(* IEC 61131-3 sources: pandora_hardware/epos_controller, 7 files *)

(* ---- canRecover.TYP ---- *)
[IEC_IEC_NORM]
TYPE CAN_RECOVER_STATE :(
	CAN_CanError,
	CAN_PowerOffGracefully,
	CAN_Sleep,
	CAN_CanReset,
	CAN_CanReset_loop,
	CAN_SleepWait
) := CAN_CanError;
END_TYPE

(* ---- initial.TYP ---- *)
[IEC_IEC_NORM]
TYPE INITIALIZE_STATE :(
	(*Initialize all axis*)
	INITIALIZE_Init,		(* 0 *)
	(*check the status of axis0*)
	INITIALIZE_CheckAxis0,	(* 1 *)
	(*check the status of axis1*)
	INITIALIZE_CheckAxis1,	(* 2 *)
	(*check the status of axis2*)
	INITIALIZE_CheckAxis2,  (* 3 *)
	(*check the status of axis3*)
	INITIALIZE_CheckAxis3,  (* 4 *)
	(*power of both axis*)
	INITIALIZE_PowerOff,	(* 5 *)
	(*reset axis0*)
	INITIALIZE_Reset0,		(* 6 *)
	(*loop until axis0 is reset*)
	INITIALIZE_Reset0_loop,	(* 7 *)
	(*reset axis1*)
	INITIALIZE_Reset1,		(* 8 *)
	(*wait until axis1 is reset*)
	INITIALIZE_Reset1_loop,	(* 9 *)
	(*reset axis2*)
	INITIALIZE_Reset2,      (* 10 *)
	(*loop until axis2 is reset*)
	INITIALIZE_Reset2_loop, (* 11 *)
	(*reset axis3*)
	INITIALIZE_Reset3,      (* 12 *)
	(*loop until axis3 is reset*)
	INITIALIZE_Reset3_loop, (* 13 *)
	(*power on all axis*)
	INITIALIZE_PowerOn,		(* 14 *)
	(*stop both axis*)
	INITIALIZE_Stop,		(* 15 *)
	(*loop until all axis have stoped*)
	INITIALIZE_Stop_loop,	(* 16 *)
	INITIALIZE_StateHalt0,	(* 17 *)
	INITIALIZE_CanError,    (* 18 *)
	INITIALIZE_CanError_loop(* 19 *)
) := INITIALIZE_Init;
END_TYPE

(* ---- initialize.TYP ---- *)
[IEC_IEC_NORM]
TYPE INITIALIZE_STATE :(
	(*Initialize both axis*)
	INITIALIZE_Init,		(* 0 *)
	(*check the status of axis0*)
	INITIALIZE_CheckAxis0,	(* 1 *)
	(*check the status of axis1*)
	INITIALIZE_CheckAxis1,	(* 2 *)
	(*power of both axis*)
	INITIALIZE_PowerOff,	(* 3 *)
	(*reset axis0*)
	INITIALIZE_Reset0,		(* 4 *)
	(*loop until axis0 is reset*)
	INITIALIZE_Reset0_loop,	(* 5 *)
	(*reset axis1*)
	INITIALIZE_Reset1,		(* 6 *)
	(*wait until axis1 is reset*)
	INITIALIZE_Reset1_loop,	(* 7 *)
	(*power on both axis*)
	INITIALIZE_PowerOn,		(* 8 *)
	(*stop both axis*)
	INITIALIZE_Stop,		(* 9 *)
	(*loop until both axis have stoped*)
	INITIALIZE_Stop_loop,	(* 10 *)
	INITIALIZE_StateHalt0,	(* 11 *)
	INITIALIZE_CanError,
	INITIALIZE_CanError_loop
) := INITIALIZE_Init;
END_TYPE

(* ---- usertype.typ ---- *)
[IEC_IEC_NORM]
TYPE MAIN_STATE :(
	(*initialize all controllers to power on - stand still*)
	(*uses function block FB_INITIALIZE*)
	MAIN_Init,					(* 0 *)
	MAIN_Init_loop,				(* 1 *)

	(*Resets the 3s timeout timer to zero*)
	MAIN_ResetTimer,			(* 2 *)

	(*Reads the control word from EPOS*)
	MAIN_Read,					(* 3 *)
	MAIN_Read_loop,				(* 4 *)

	(*Reads the actual velocity of EPOS P and stores it to a local variable*)
	MAIN_Read_Velocity,			(* 5 *)
	MAIN_Read_Velocity_loop,	(* 6 *)

	(*Reads the actual current of EPOS P and stores it to a local variable*)
	MAIN_Read_Current,			(* 7 *)
	MAIN_Read_Current_loop,		(* 8 *)

	(*Writes the actual velocity of EPOS P from the local variable to EPOS object dictionary*)
	MAIN_Write_Velocity,		(* 9 *)
	MAIN_Write_Velocity_loop,	(* 10 *)

	(*Writes the actual current of EPOS P from the local variable to EPOS object dictionary*)
	MAIN_Write_Current,			(* 11 *)
	MAIN_Write_Current_loop,	(* 12 *)

	(*updatess the timeout timer*)
	(*if the timer reaches 3s switches to state halt*)
	MAIN_UpdateTimer,			(* 13 *)

	(*Executes the move specified by the control word*)
	MAIN_StateAxis_Move,		(* 14 *)

	(*Resets the control word in order to accept a new command*)
	MAIN_StateWrite,			(* 15 *)

	(*halts all motors*)
	MAIN_StateHalt0,			(* 16 *)
	MAIN_StateHalt1,			(* 17 *)

	(*attempts an error recovery if there is CAN error*)
	(*uses function block FB_CanRecover*)
	MAIN_CanError,				(* 18 *)
	MAIN_CanError_loop,			(* 19 *)

	(*Intercepts non-CAN errors coming from other FBs to MAIN_Init*)
	(*uses FB_ErrorWarning to write error codes to EPOS Object Dictionary*)
	MAIN_Error,					(* 20 *)
	MAIN_Error_loop				(* 21 *)
	) := MAIN_Init;
END_TYPE

TYPE INITIALIZE_STATE :(
	(*Initialize both axis*)
	INITIALIZE_Init,		(* 0 *)
	(*check the status of axis0*)
	INITIALIZE_CheckAxis0,	(* 1 *)
	(*check the status of axis1*)
	INITIALIZE_CheckAxis1,	(* 2 *)
	(*check the status of axis2*)
	INITIALIZE_CheckAxis2,  (* 3 *)
	(*check the status of axis3*)
	INITIALIZE_CheckAxis3,  (* 4 *)
	(*power of both axis*)
	INITIALIZE_PowerOff,	(* 5 *)
	(*reset axis0*)
	INITIALIZE_Reset0,		(* 6 *)
	(*loop until axis0 is reset*)
	INITIALIZE_Reset0_loop,	(* 7 *)
	(*reset axis1*)
	INITIALIZE_Reset1,		(* 8 *)
	(*wait until axis1 is reset*)
	INITIALIZE_Reset1_loop,	(* 9 *)
	(*reset axis2*)
	INITIALIZE_Reset2,      (* 10 *)
	(*loop until axis2 is reset*)
	INITIALIZE_Reset2_loop, (* 11 *)
	(*reset axis3*)
	INITIALIZE_Reset3,      (* 12 *)
	(*loop until axis3 is reset*)
	INITIALIZE_Reset3_loop, (* 13 *)
	(*power on all axis*)
	INITIALIZE_PowerOn,		(* 14 *)
	(*stop all axis*)
	INITIALIZE_Stop,		(* 15 *)
	(*loop until all axis have stoped*)
	INITIALIZE_Stop_loop,	(* 16 *)
	INITIALIZE_StateHalt0,	(* 17 *)
	INITIALIZE_CanError,    (* 18 *)
	INITIALIZE_CanError_loop(* 19 *)
) := INITIALIZE_Init;
END_TYPE

(* ---- FB_CanRecover.ST ---- *)
FUNCTION_BLOCK FB_CanRecover
VAR_EXTERNAL
	Axis0 				                    : Axis_REF;
	Axis1 				                    : Axis_REF;
	Axis2                                   : Axis_REF;
	Axis3                                   : Axis_REF;
END_VAR

VAR_INPUT
	Execute : BOOL;
END_VAR

VAR_OUTPUT
    Done                      : BOOL;
    Error                     : BOOL;
	ErrorID                   : DINT;
END_VAR

VAR
	lastErrorId : DINT :=0;
	internalErrorCounter : UDINT := 0;
	canState	: CAN_RECOVER_STATE;

	fbPower0 : MC_Power;
	fbPower1 : MC_Power;
	fbPower2 : MC_Power;
	fbPower3 : MC_Power;

	fbTimer : TON;

	fbReset0 : MC_Reset;
	fbReset1 : MC_Reset;
	fbReset2 : MC_Reset;
	fbReset3 : MC_Reset;

END_VAR
IF Execute = FALSE THEN

	Done:=FALSE;
	lastErrorId:=0;
	internalErrorCounter:=0;
	canState:=CAN_CanError;

ELSE

	IF canState = CAN_CanError THEN

		IF internalErrorCounter > 5 THEN

			Error := TRUE;
			ErrorId := LastErrorId;
		ELSE

			canState := CAN_PowerOffGracefully;
		END_IF;

	ELSIF canState = CAN_PowerOffGracefully THEN
		(*attempt to stop all controllers*)

		(*Disable power on all controllers*)
		fbPower0(Axis := Axis0 , Enable := FALSE);
		fbPower1(Axis := Axis1 , Enable := FALSE);
		fbPower2(Axis := Axis2 , Enable := FALSE);
		fbPower3(Axis := Axis3 , Enable := FALSE);

		(*Switch state when all controllers are disabled*)
		(*or have an error*)
		IF ( ( NOT fbPower0.Status ) OR fbPower0.Error ) AND
	       ( ( NOT fbPower1.Status ) OR fbPower1.Error ) AND
		   ( ( NOT fbPower2.Status ) OR fbPower2.Error ) AND
	       ( ( NOT fbPower3.Status ) OR fbPower3.Error ) THEN
			(*all controllers are disabled or in an error state, switch to the next state*)
			canState := CAN_Sleep;
		END_IF;

	ELSIF canState = CAN_Sleep THEN

		fbTimer(In := false , Pt := t#1s);
		canState := CAN_SleepWait;

	ELSIF canState = CAN_SleepWait THEN

		fbTimer(In := true , Pt := t#1s);

		IF fbTimer.Q THEN
			canState := CAN_CanReset;
		END_IF;

	ELSIF canState = CAN_CanReset THEN

		fbReset0(Axis := Axis0 , Execute := FALSE);
		fbReset1(Axis := Axis1 , Execute := FALSE);
		fbReset2(Axis := Axis2 , Execute := FALSE);
		fbReset3(Axis := Axis3 , Execute := FALSE);
		canState := CAN_CanReset_loop;

	ELSIF canState = CAN_CanReset_loop THEN

		fbReset0(Axis := Axis0 , Execute := TRUE);
		fbReset1(Axis := Axis1 , Execute := TRUE);
		fbReset2(Axis := Axis2 , Execute := TRUE);
		fbReset3(Axis := Axis3 , Execute := TRUE);

		IF fbReset0.Error OR fbReset1.Error THEN

			IF fbReset0.Error THEN
				lastErrorId := fbReset0.ErrorId;
			ELSE
				lastErrorId := fbReset1.ErrorId;
			END_IF;

			internalErrorCounter := internalErrorCounter +1;
			canState :=CAN_CanError;

		ELSIF fbReset0.DONE AND fbReset1.DONE THEN
			Done := TRUE;
			(*canState := CAN_Init;*)
		END_IF;
	END_IF;

END_IF;

END_FUNCTION_BLOCK

(* ---- FB_INITIALIZE.ST ---- *)
FUNCTION_BLOCK FB_INITIALIZE
VAR_EXTERNAL
	Axis0 				                    : Axis_REF;                    (* Axis definitions, Node 2, Right Wheel, EPOS controller *)
	Axis1 				                    : Axis_REF;					   (* Axis definitions, Node 1, Left Wheel *)
END_VAR

VAR_INPUT
	Execute : BOOL;
END_VAR

VAR_OUTPUT
    Done                      : BOOL;
    Error                     : BOOL;
	ErrorID                   : DINT;
END_VAR

VAR
	lastErrorId : DINT :=0;
	internalErrorCounter : UDINT := 0;
	initializationState	: INITIALIZE_STATE;

	fbReadStatus0	: MC_ReadStatus;
	fbReadStatus1	: MC_ReadStatus;

	fbPower0		: MC_Power;
	fbPower1		: MC_Power;

	fbAxisStop0		: MC_Stop;
	fbAxisStop1		: MC_Stop;

	fbReset0		: MC_Reset;
	fbReset1		: MC_Reset;

	fbCanRecover 	: FB_CanRecover;

END_VAR
IF Execute = FALSE THEN

	initializationState := INITIALIZE_Init;
	Done := FALSE;
	Error := FALSE;
	ErrorId := 0;
	internalErrorCounter := 0;

ELSE

	IF initializationState = INITIALIZE_Init THEN

		IF internalErrorCounter >= 5 THEN

			Error := TRUE;
			ErrorId := lastErrorId;
			Done := FALSE;

		ELSE

			(*initialize both controllers to velocity mode, stand still*)

			fbReadStatus0(Axis := Axis0 , Enable := TRUE);
			fbReadStatus1(Axis := Axis1 , Enable := TRUE);

			IF fbReadStatus0.Error OR fbReadStatus1.Error THEN

				(*cannot read the state of one or both controllers*)
				(*go to state canError to check for errors*)

				(*initializationState := MAIN_CanError;*)
				initializationState := INITIALIZE_CanError;

			ELSIF fbReadStatus0.Valid AND fbReadStatus1.Valid THEN

				(*function blocks fbReadStatus0/1 have updated their values*)
				IF fbReadStatus0.Disabled AND fbReadStatus1.Disabled THEN

					(*both controllers are disabled*)
					(*switch to state INITIALIZE_PowerOn to enable them*)
					initializationState := INITIALIZE_PowerOn;

				ELSIF NOT fbReadStatus0.Disabled THEN

					(*axis 0 - EPOS controller - Node 2 - right motor is not disabled*)
					(*switch to state INITIALIZE_CheckAxis0 to disable it*)

					initializationState := INITIALIZE_CheckAxis0;

				ELSIF NOT fbReadStatus1.Disabled THEN

					(*axis 1 - EPOS controller - Node 1 - left motor is not disabled*)
					(*switch to state INITIALIZE_CheckAxis1 to disable it*)

					initializationState := INITIALIZE_CheckAxis1;

				END_IF;

			ELSE

				(*the fbReadStatus0/1 blocks have not updated their values yet*)
				(*continue calling them with enable:=TRUE until they do*)
				(*no need to change state*)
				;

			END_IF;

		END_IF;

	ELSIF initializationState = INITIALIZE_CheckAxis0 THEN

		(*check the state of Axis0*)
		(*after the sequence completes the axis will be in the disabled state*)
		(*control is transfered to state INITIALIZE_Init that will start the enable sequence*)

	    fbReadStatus0(Axis := Axis0 , Enable := TRUE);

		IF fbReadStatus0.Error THEN

			(*cannot read the status of axis0*)
			(*axis0 is the EPOS controller connected on the CAN bus*)
			(*maybe there is a CAN communication error, switch to state MAIN_CanError*)
			(*initializationState := MAIN_CanError;*)
			initializationState := INITIALIZE_CanError;

		ELSIF fbReadStatus0.Valid THEN

			(*we have read the status of axis0*)

			IF fbReadStatus0.Errorstop THEN
				(*the motor is in an error state*)
				(*call the MC_Reset function block to reset it*)
				initializationState := INITIALIZE_Reset0;
			ELSIF fbReadStatus0.Disabled THEN
				(*the motor is in the disabled state, nothing to do*)
				(*switch to MAIN_Init*)
				initializationState := INITIALIZE_Init;
			ELSIF fbReadStatus0.Stopping THEN
				(*the motor is stopping*)
				(*although we could simply wait, force the stop*)
				(*i.e. greater decceleration*)
				initializationState := INITIALIZE_Reset0;
			ELSIF fbReadStatus0.StandStill THEN
				(*the controller is not in an error state but it is enabled*)
				(*power off both controllers*)
				initializationState := INITIALIZE_PowerOff;
			ELSIF fbReadStatus0.DiscreteMotion THEN
				(*i.e. position control*)
				(*stop motion on both controllers*)
				initializationState := INITIALIZE_Stop;
			ELSIF fbReadStatus0.ContinuousMotion THEN
				(*i.e. velocity control*)
				(*stop motion on both controllers*)
				initializationState := INITIALIZE_Stop;
			ELSIF fbReadStatus0.Homing THEN
				(*stop homing on both controllers*)
				initializationState := INITIALIZE_Stop;
			END_IF;
		ELSE
			(*status not updated yet*)
			;
		END_IF;

	ELSIF initializationState = INITIALIZE_CheckAxis1 THEN

		(*check the state of Axis1*)
		(*after the sequence completes the axis will be in the disabled state*)
		(*control is transfered to state MAIN_Init that will start the enable sequence*)

	    fbReadStatus1(Axis := Axis1 , Enable := TRUE);

		IF fbReadStatus1.Error THEN

			(*this is wierd*)
			(*there is no reason why we cannot read our own status*)
			(*axis1 is the EPOS P controller*)
			(*simply increment the internal error counter and try again*)
			lastErrorId := fbReadStatus1.ErrorId;
			internalErrorCounter := internalErrorCounter + 1;
			initializationState := INITIALIZE_Init;

		ELSIF fbReadStatus1.Valid THEN
			(*we have read the status of axis1*)

			IF fbReadStatus1.Errorstop THEN
				(*the motor is in an error state*)
				(*call the MC_Reset function block to reset it*)
				initializationState := INITIALIZE_Reset1;
			ELSIF fbReadStatus1.Disabled THEN
				(*the motor is in the disabled state, nothing to do*)
				(*switch to MAIN_Init*)
				initializationState := INITIALIZE_Init;
			ELSIF fbReadStatus1.Stopping THEN
				(*the motor is stopping*)
				(*although we could simply wait, force the stop*)
				(*i.e. greater decceleration*)
				initializationState := INITIALIZE_Reset1;
			ELSIF fbReadStatus1.StandStill THEN
				(*the controller is not in an error state but it is enabled*)
				(*power off both controllers*)
				initializationState := INITIALIZE_PowerOff;
			ELSIF fbReadStatus1.DiscreteMotion THEN
				(*i.e. position control*)
				(*stop motion on both controllers*)
				initializationState := INITIALIZE_Stop;
			ELSIF fbReadStatus1.ContinuousMotion THEN
				(*i.e. velocity control*)
				(*stop motion on both controllers*)
				initializationState := INITIALIZE_Stop;
			ELSIF fbReadStatus1.Homing THEN
				(*stop homing on both controllers*)
				initializationState := INITIALIZE_Stop;
			END_IF;
		ELSE
			(*status not updated yet*)
			;
		END_IF;

	ELSIF initializationState = INITIALIZE_PowerOff THEN

		(*Disable power on both controllers*)
		fbPower0(Axis := Axis0 , Enable := FALSE);
		fbPower1(Axis := Axis1 , Enable := FALSE);

		(*Switch state when both controllers are disabled*)
		IF fbPower0.Error OR fbPower1.Error THEN

			initializationState := INITIALIZE_Init;

		ELSIF ( NOT fbPower0.Status ) AND ( NOT fbPower1.Status ) THEN
			(*both controllers are disabled, switch to the next state*)
			initializationState := INITIALIZE_Init;
		END_IF;

	ELSIF initializationState = INITIALIZE_Reset0 THEN

		(*reset axis0*)

		fbReset0(Axis := Axis0 , Execute := FALSE);
		initializationState := INITIALIZE_Reset0_loop;

	ELSIF initializationState = INITIALIZE_Reset0_loop THEN

		fbReset0(Axis := Axis0 , Execute := TRUE);

		IF fbReset0.ERROR THEN
			(*check for can communication errors*)
			(*initializationState := MAIN_CanError;*)
			initializationState := INITIALIZE_CanError;
			;
		ELSIF fbReset0.DONE THEN
			(*done reseting*)
			initializationState := INITIALIZE_Init;
		END_IF;

	ELSIF initializationState = INITIALIZE_Reset1 THEN

		(*reset axis1*)

		fbReset1(Axis := Axis1 , Execute := FALSE);
		initializationState := INITIALIZE_Reset1_loop;

	ELSIF initializationState = INITIALIZE_Reset1_loop THEN

		fbReset1(Axis := Axis1 , Execute := TRUE);

		IF fbReset1.ERROR THEN

			(*this is wierd*)
			(*there is no reason why we cannot reset our controller*)
			(*axis1 is the EPOS P controller*)
			(*simply increment the internal error counter and try again*)
			internalErrorCounter := internalErrorCounter + 1;
			initializationState := INITIALIZE_Init;

		ELSIF fbReset1.DONE THEN
			(*done reseting*)
			initializationState := INITIALIZE_Init;
		END_IF;

	ELSIF initializationState = INITIALIZE_Stop THEN

		(*stop both axis*)

		fbAxisStop0(Axis := Axis0, Execute := FALSE, Deceleration := 10000);
		fbAxisStop1(Axis := Axis1, Execute := FALSE, Deceleration := 10000);
		initializationState := INITIALIZE_Stop_loop;

	ELSIF initializationState = INITIALIZE_Stop_loop THEN

		fbAxisStop0(Axis := Axis0, Execute := TRUE, Deceleration := 10000);
		fbAxisStop1(Axis := Axis1, Execute := TRUE, Deceleration := 10000);

		IF fbAxisStop0.Error OR fbAxisStop1.Error THEN

			(*ther is an error while attempting to stop one, or both of the controllers*)
			(*re-initialize the controllers*)
			initializationState:=INITIALIZE_Init;

		ELSIF fbAxisStop0.Done AND fbAxisStop1.DONE THEN
			(*both controllers have stopped*)
			(*switch to state init*)
			initializationState := INITIALIZE_Init;

		END_IF;

	ELSIF initializationState = INITIALIZE_PowerOn THEN

		(*power on both controllers*)

		fbPower0(Axis := Axis0, Enable := TRUE);
		fbPower1(Axis := Axis1, Enable := TRUE);

		IF fbPower0.Error OR fbPower1.Error THEN
			(*ther is an error while attempting to power on one, or both of the controllers*)
			(*re-initialize the controllers*)
			initializationState:=INITIALIZE_Init;
		ELSIF fbPower0.Status AND fbPower1.Status THEN
			(*both controllers are powered on*)
			(*go start the control sequence*)
			Done := TRUE;
		END_IF;
	ELSIF initializationState = INITIALIZE_CanError THEN

		fbCanRecover(Execute:=FALSE);
		initializationState := INITIALIZE_CanError_loop;

	ELSIF initializationState = INITIALIZE_CanError_loop THEN
		fbCanRecover(Execute:=TRUE);
		IF fbCanRecover.Error THEN

			lastErrorId:=fbCanRecover.ErrorId;
			internalErrorCounter := internalErrorCounter + 1;
			initializationState := INITIALIZE_Init;

		ELSIF fbCanRecover.Done THEN
			initializationState := INITIALIZE_Init;
		END_IF;
	END_IF;
END_IF;

END_FUNCTION_BLOCK

(* ---- PROG_MAIN.ST ---- *)
PROGRAM PROG_MAIN
VAR_EXTERNAL
    Axis0                 : Axis_REF;   (*Right_back wheel Node 2,communication*)
    Axis1                 : Axis_REF;   (*Right_front wheel Node 1,EPOSP*)
    Axis2                 : Axis_REF;   (*Left_back wheel Node 3*)
    Axis3                 : Axis_REF;   (*Left_front wheel Node 4*)

END_VAR

VAR_GLOBAL

END_VAR

VAR

   	fbPower0							: MC_Power;
	fbPower1							: MC_Power;
	fbPower2							: MC_Power;
	fbPower3							: MC_Power;
	fbReset0							: MC_Reset;
	fbReset1							: MC_Reset;
	fbReset2							: MC_Reset;
	fbReset3							: MC_Reset;

	fbReadStatus0						: MC_ReadStatus;
	fbReadStatus1						: MC_ReadStatus;
	fbReadStatus2						: MC_ReadStatus;
	fbReadStatus3						: MC_ReadStatus;

	fbReadActualVelocity0				: MC_ReadActualVelocity;
	fbReadActualVelocity1				: MC_ReadActualVelocity;
	fbReadActualVelocity2				: MC_ReadActualVelocity;
	fbReadActualVelocity3				: MC_ReadActualVelocity;

	fbReadActualCurrent0				: MC_ReadActualCurrent;
	fbReadActualCurrent1				: MC_ReadActualCurrent;
	fbReadActualCurrent2				: MC_ReadActualCurrent;
	fbReadActualCurrent3				: MC_ReadActualCurrent;

	fbAxisMove0              			: MC_MoveVelocity;
	fbAxisStop0							: MC_Stop;
	fbAxisMove1              			: MC_MoveVelocity;
	fbAxisStop1							: MC_Stop;
	fbAxisMove2              			: MC_MoveVelocity;
	fbAxisStop2							: MC_Stop;
	fbAxisMove3              			: MC_MoveVelocity;
	fbAxisStop3							: MC_Stop;

	fbReadObject						: FB_MAIN_StateRead;
	fbWriteObject						: FB_MAIN_StateWrite;

	fbGetObjectEncoder		  			: MU_GetObject;
	fbSetObjectEncoder		  			: MU_SetObject;

	fbTimer								: TON;

	extractedValue						: UDINT := 0;
	velByte1							: UDINT;
	velByte2							: UDINT;
	leftSign							: UDINT;
	leftVeloc							: UDINT;
	freshByte							: UDINT;
	rightSign							: UDINT;
	rightVeloc							: UDINT;

	maxVelocity							: UDINT := 5500;

	udEncoderTemp						: UDINT := 0;
	dEncoderValue						: DINT := 0;

	oExecuteReset0						: BOOL;
	oExecuteReset1						: BOOL;
	oExecutePower0						: BOOL;
	oExecutePower1						: BOOL;

	oExecuteTimerStart					: BOOL;
	oExecuteObjectReading				: BOOL;
	oExecuteObjectWriting				: BOOL;

	oExecuteObjectReadingEncoder		: BOOL;
	oExecuteObjectWritingEncoder		: BOOL;
	oExecuteAxisMove					: BOOL;

	fbGetVelocity			: MU_GetObject;
	fbGetCurrent			: MU_GetObject;
    fbWriteVelocity			: MU_SetObject;
	fbWriteCurrent			: MU_SetObject;

	velocityActualValue : UDINT;
	currentActualValue : UDINT;
	internalErrorCounter : UDINT;

	fbInitialize : FB_INITIALIZE;
	fbCanRecover : FB_CanRecover;

END_VAR
IF eStateMain = MAIN_Init THEN;
    fbInitialize(Execute := FALSE);
	eStateMain := MAIN_Init_loop;
ELSIF eStateMain = MAIN_Init_loop THEN
    fbInitialize(Execute := TRUE);
	IF fbInitialize.Error THEN  	(*Hope, this never happens...*)
	    eStateMain := MAIN_Init;
	ELSIF fbInitialize.Done THEN
	    eStateMain := MAIN_ResetTimer;
	END_IF;
ELSIF eStateMain = MAIN_ResetTimer THEN

    (*reset the timer back to zero*)

    fbTimer (In := false, Pt := t#3s);

	(*read axis1 actual velocity*)

	eStateMain := MAIN_Read_Velocity;

(*Read from EPOSP velocity from 2028 Axis 1 EPOSP*)

ELSIF eStateMain = MAIN_Read_Velocity THEN
    fbGetVelocity(Axis := Axis1, Enable := FALSE, Index := 16#2028 , Subindex := 16#00);
	eStateMain := MAIN_Read_Velocity_loop;
ELSIF eStateMain = MAIN_Read_Velocity_loop THEN

	fbGetVelocity(Axis := Axis1, Enable := TRUE, Index := 16#2028, Subindex := 16#00);
	IF (fbGetVelocity.Error) THEN
	    internalErrorCounter := internalErrorCounter + 1;
		eStateMain := MAIN_Init;
	ELSIF (fbGetVelocity.Done) THEN
	    velocityActualValue := fbGetVelocity.Value;  (*store velocity actual value to a global variable*)
        IF (velocityActualValue>2147483647) then
		    velocityActualValue := velocityActualValue+20000;
		END_IF;
		eStateMain := MAIN_Write_Velocity;
	END_IF;

(*write EPOSP velocity to 206B register of epos-axis0 in order to read it There is no communication between PC and EPOSP *)

ELSIF eStateMain = MAIN_Write_Velocity THEN
    fbWriteVelocity(Axis := Axis0, Execute := FALSE, Index := 16#206B, Subindex := 16#00, Value:= velocityActualValue);

	eStateMain := MAIN_Write_Velocity_loop;

ELSIF eStateMain = MAIN_Write_Velocity_loop THEN
	fbWriteVelocity(Axis := Axis0, Execute := TRUE, Index := 16#206B, Subindex := 16#00, Value:= velocityActualValue);

	IF fbWriteVelocity.Error THEN
	    eStateMain := MAIN_CanError;
	ELSIF fbWriteVelocity.Done THEN
	    eStateMain := MAIN_Read_Current;
	END_IF;

(*Read EPOSP (axis 1) current from register 2027*)

ELSIF eStateMain = MAIN_Read_Current THEN
    fbGetCurrent (Axis := Axis1, Enable := FALSE, Index := 16#2027 , Subindex := 16#00);
	eStateMain := MAIN_Read_Current_loop;

ELSIF eStateMain = MAIN_Read_Current_loop THEN
    fbGetCurrent (Axis := Axis1, Enable := true, Index := 16#2027 , Subindex := 16#00);
	IF fbGetCurrent.Error THEN
	    eStateMain := MAIN_Init;
	ELSIF fbGetCurrent.Done THEN
	    currentActualValue := fbGetCurrent.Value;
		IF (currentActualValue>2147483647) THEN
		    currentActualValue := currentActualValue + 20000;
		END_IF;
		eStateMain := MAIN_Write_Current;
	END_IF;

(*Write EPOSP current to 2030 register of epos communication (axis0)*)

ELSIF eStateMain = MAIN_Write_Current THEN
    fbWriteCurrent(Axis := Axis0, Execute := FALSE, Index := 16#2030, Subindex := 16#00, Value:= currentActualValue);

	eStateMain := MAIN_Write_Current_loop;

ELSIF eStateMain = MAIN_Write_Current_loop THEN
    fbWriteCurrent(Axis := Axis0, Execute := TRUE, Index := 16#2030, Subindex := 16#00, Value:= currentActualValue);

    IF (fbWriteCurrent.Error) THEN
	    eStateMain := MAIN_Init;
	ELSIF (fbWriteCurrent.Done) THEN
	    eStateMain := MAIN_Read;
	END_IF;

ELSIF eStateMain = MAIN_Read THEN
     (*read the control word from EPOS*)

	 fbReadObject (Axis := Axis0, Execute := FALSE);
	 eStateMain := MAIN_Read_loop;

ELSIF eStateMain = MAIN_Read_loop THEN
    fbReadObject (Axis := Axis0, Execute := TRUE);
	IF (fbReadObject.Error) THEN
	    eStateMain := MAIN_Init;

	ELSIF fbReadObject.Done AND fbReadObject.Done1 THEN
	(*Velocity Fresh*)

	    extractedValue := fbReadObject.velocityWord;

		(* Low Byte *)
		velByte1 := extractedValue MOD 16#00010000;
		leftSign := ( velByte1 / 16#00004000 ) MOD 16#00000002;
		leftVeloc := velByte1 MOD 16#00004000;

		(* High Byte *)
		velByte2 := extractedValue / 16#00010000;
		rightSign := ( velByte2 / 16#00004000 ) MOD 16#00000002;
		rightVeloc := velByte2 MOD 16#00004000;
		eStateMain := MAIN_StateWrite;

		fbTimer(In := false , Pt := t#3s);

	ELSIF fbReadObject.Done THEN
		eStateMain := MAIN_UpdateTimer;
	END_IF;

ELSIF eStateMain = MAIN_UpdateTimer THEN

	fbTimer(In := TRUE , Pt := t#3s);

	IF fbTimer.Q THEN
		eStateMain := MAIN_StateHalt0;
	ELSE
		eStateMain := MAIN_Read_Velocity;
	END_IF;

ELSIF eStateMain = MAIN_StateWrite THEN

	  fbWriteObject(Axis := Axis0, Execute := oExecuteObjectWriting, CurrentValue := extractedValue);
	  oExecuteObjectWriting := TRUE;

	  IF fbWriteObject.Done AND (NOT fbWriteObject.Error) THEN
	        oExecuteObjectWriting := FALSE;

			fbAxisMove0(Axis := Axis0, Execute := FALSE, Velocity := 1000 , Acceleration := 100 , Deceleration := 100 , Direction := MCpositive);
        	fbAxisMove1(Axis := Axis1, Execute := FALSE, Velocity := 1000 , Acceleration := 100 , Deceleration := 100 , Direction := MCpositive);
			fbAxisMove2(Axis := Axis2, Execute := FALSE, Velocity := 1000 , Acceleration := 100 , Deceleration := 100 , Direction := MCpositive);
        	fbAxisMove3(Axis := Axis3, Execute := FALSE, Velocity := 1000 , Acceleration := 100 , Deceleration := 100 , Direction := MCpositive);
			fbAxisStop0(Axis := Axis0, Execute := FALSE);
			fbAxisStop1(Axis := Axis1, Execute := FALSE);
			fbAxisStop2(Axis := Axis2, Execute := FALSE);
			fbAxisStop3(Axis := Axis3, Execute := FALSE);
			fbWriteObject(Axis := Axis0, Execute := FALSE);
			fbWriteObject(Axis := Axis2, Execute := FALSE);
			fbWriteObject(Axis := Axis3, Execute := FALSE);
			oExecuteAxisMove := FALSE;
	        eStateMain := MAIN_StateAxis_Move;
	  END_IF;

ELSIF eStateMain = MAIN_StateHalt0 THEN

	fbAxisStop0(Axis := Axis0 , Execute := FALSE , Deceleration := 10000);
	fbAxisStop1(Axis := Axis1 , Execute := FALSE , Deceleration := 10000);
	fbAxisStop2(Axis := Axis2 , Execute := FALSE , Deceleration := 10000);
	fbAxisStop3(Axis := Axis3 , Execute := FALSE , Deceleration := 10000);

	eStateMain := MAIN_StateHalt1;

ELSIF eStateMain = MAIN_StateHalt1 THEN

	fbReadStatus0(Axis := Axis0 , Enable := TRUE);
	fbReadStatus1(Axis := Axis1 , Enable := TRUE);
	fbReadStatus2(Axis := Axis2 , Enable := TRUE);
	fbReadStatus3(Axis := Axis3 , Enable := TRUE);

	IF fbReadStatus0.Error OR fbReadStatus1.Error OR fbReadStatus2.Error OR fbReadStatus3.Error THEN

		(*cannot read the state of 1 or 2 or 3 or 4 controllers*)
		(*go to state canError to check for errors*)
		eStateMain := MAIN_CanError;

	ELSIF fbReadStatus0.Valid AND fbReadStatus1.Valid AND fbReadStatus2.Valid AND fbReadStatus3.Valid THEN

		IF fbAxisStop0.Error THEN
			eStateMain := MAIN_CanError;
		ELSIF NOT fbReadStatus0.StandStill THEN
			fbAxisStop0(Axis := Axis0 , Execute := TRUE , Deceleration := 10000);
		END_IF;

		IF fbAxisStop1.Error THEN
			eStateMain := MAIN_CanError;
		ELSIF NOT fbReadStatus1.StandStill THEN
			fbAxisStop1(Axis := Axis1 , Execute := TRUE , Deceleration := 10000);
		END_IF;
		IF fbAxisStop2.Error THEN
			eStateMain := MAIN_CanError;
		ELSIF NOT fbReadStatus2.StandStill THEN
			fbAxisStop2(Axis := Axis2 , Execute := TRUE , Deceleration := 10000);
		END_IF;

		IF fbAxisStop3.Error THEN
			eStateMain := MAIN_CanError;
		ELSIF NOT fbReadStatus3.StandStill THEN
			fbAxisStop3(Axis := Axis3 , Execute := TRUE , Deceleration := 10000);
		END_IF;

		IF fbReadStatus0.StandStill AND fbReadStatus1.StandStill AND fbReadStatus2.StandStill AND fbReadStatus3.StandStill THEN

			oExecuteAxisMove := FALSE;
		  	eStateMain := MAIN_ResetTimer;

		END_IF;

	END_IF;

ELSIF eStateMain = MAIN_StateAxis_Move THEN

	  (* Limiter *)
	  IF (leftVeloc > maxVelocity) THEN
	  	leftVeloc := maxVelocity;
	  END_IF;

	  (* Limiter *)
	  IF (rightVeloc > maxVelocity) THEN
	  	rightVeloc := maxVelocity;
	  END_IF;

	  IF (rightVeloc = 0) THEN
	  	fbAxisStop0(Axis := Axis0 , Execute := oExecuteAxisMove , Deceleration := 10000);
	  ELSIF (rightSign = 1) THEN
      	fbAxisMove0(Axis := Axis0, Execute := oExecuteAxisMove, Velocity := rightVeloc,
                Acceleration := 10000, Deceleration := 10000,
				Direction := MCnegative);
	  ELSE
	  	fbAxisMove0(Axis := Axis0, Execute := oExecuteAxisMove, Velocity := rightVeloc,
                Acceleration := 10000, Deceleration := 10000,
				Direction := MCpositive);
	  END_IF;

	  IF (rightVeloc = 0) THEN
	  	fbAxisStop1(Axis := Axis1 , Execute := oExecuteAxisMove , Deceleration := 10000);
	  ELSIF (rightsign = 1) THEN
	  	fbAxisMove1(Axis := Axis1, Execute := oExecuteAxisMove, Velocity := rightVeloc,
                Acceleration := 10000, Deceleration := 10000,
				Direction := MCnegative);
	  ELSE
	  	fbAxisMove1(Axis := Axis1, Execute := oExecuteAxisMove, Velocity := rightVeloc ,Acceleration := 10000, Deceleration := 10000, Direction := MCpositive);
	  END_IF;

	  IF (leftVeloc = 0) THEN
	  	fbAxisStop2(Axis := Axis2 , Execute := oExecuteAxisMove , Deceleration := 10000);
	  ELSIF (leftSign = 1) THEN
      	fbAxisMove2(Axis := Axis2, Execute := oExecuteAxisMove, Velocity := leftVeloc,
                Acceleration := 10000, Deceleration := 10000,
				Direction := MCnegative);
	  ELSE
	  	fbAxisMove2(Axis := Axis2, Execute := oExecuteAxisMove, Velocity := leftVeloc,
                Acceleration := 10000, Deceleration := 10000,
				Direction := MCpositive);
	  END_IF;

	  IF (leftVeloc = 0) THEN
	  	fbAxisStop3(Axis := Axis3 , Execute := oExecuteAxisMove , Deceleration := 10000);
	  ELSIF (leftsign = 1) THEN
	  	fbAxisMove3(Axis := Axis3, Execute := oExecuteAxisMove, Velocity := leftVeloc,
                Acceleration := 10000, Deceleration := 10000,
				Direction := MCnegative);
	  ELSE
	  	fbAxisMove3(Axis := Axis3, Execute := oExecuteAxisMove, Velocity := leftVeloc ,Acceleration := 10000, Deceleration := 10000, Direction := MCpositive);
	  END_IF;

	  oExecuteAxisMove := TRUE;

	  fbReadStatus0(Axis := Axis0 , Enable := TRUE);
	  fbReadStatus1(Axis := Axis1 , Enable := TRUE);
	  fbReadStatus2(Axis := Axis2 , Enable := TRUE);
	  fbReadStatus3(Axis := Axis3 , Enable := TRUE);

	  fbReadActualVelocity0(Axis := Axis0 , Enable := TRUE);
	  fbReadActualVelocity1(Axis := Axis1 , Enable := TRUE);
	  fbReadActualVelocity2(Axis := Axis2 , Enable := TRUE);
	  fbReadActualVelocity3(Axis := Axis3 , Enable := TRUE);

	  fbReadActualCurrent0(Axis := Axis0 , Enable := TRUE);
	  fbReadActualCurrent1(Axis := Axis1 , Enable := TRUE);
	  fbReadActualCurrent2(Axis := Axis2 , Enable := TRUE);
	  fbReadActualCurrent3(Axis := Axis3 , Enable := TRUE);

	  IF fbAxisMove0.Error THEN
	  	eStateMain := MAIN_Init;
	  ELSIF fbAxisStop0.Error THEN
	  	eStateMain := MAIN_Init;
	  ELSIF fbAxisMove1.Error THEN
	  	eStateMain := MAIN_Init;
	  ELSIF fbAxisStop1.Error THEN
	  	eStateMain := MAIN_Init;
	  IF fbAxisMove2.Error THEN
	  	eStateMain := MAIN_Init;
	  ELSIF fbAxisStop2.Error THEN
	  	eStateMain := MAIN_Init;
	  ELSIF fbAxisMove3.Error THEN
	  	eStateMain := MAIN_Init;
	  ELSIF fbAxisStop3.Error THEN
	  	eStateMain := MAIN_Init;
	  ELSIF (fbAxisMove0.InVelocity OR fbAxisStop0.Done ) AND (fbAxisMove1.InVelocity OR fbAxisStop1.Done ) AND
	        (fbAxisMove2.InVelocity OR fbAxisStop2.Done ) AND (fbAxisMove3.InVelocity OR fbAxisStop3.Done ) AND
	  			fbReadStatus0.Valid AND (fbReadStatus0.ContinuousMotion OR fbReadStatus0.StandStill) AND
				fbReadStatus1.Valid AND (fbReadStatus1.ContinuousMotion OR fbReadStatus1.StandStill) AND
				fbReadStatus2.Valid AND (fbReadStatus2.ContinuousMotion OR fbReadStatus2.StandStill) AND
				fbReadStatus3.Valid AND (fbReadStatus3.ContinuousMotion OR fbReadStatus3.StandStill) THEN

		oExecuteAxisMove := FALSE;
	  	eStateMain := MAIN_Read_Velocity;
	  END_IF;

ELSIF eStateMain = MAIN_CanError THEN

	fbCanRecover(Execute:=FALSE);
	eStateMain := MAIN_CanError_loop;

ELSIF eStateMain = MAIN_CanError_loop THEN

	fbCanRecover(Execute:=TRUE);
	IF fbCanRecover.Done THEN
		eStateMain:=MAIN_Init;
	END_IF;

END_IF;

END_IF;

END_PROGRAM
